# B&R Automation Studio project test
Automation Studio 4.2.5.388

## Logical view

Binary libraries used (declarations not repeated): operator, runtime, astime, AsIecCon, standard

### Global.var - Global variables
```iecst
VAR
	var2 : BOOL;
	var3 : BOOL;
	var4 : BOOL;
	var1 : BOOL;
END_VAR
```


### Program Logical/Program (IEC)

#### Cyclic.fbd - Cyclic code
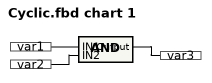
Diagram, in the editor's own instruction-list form stored in the file:
```il
PROGRAM _CYCLIC
VAR
	zz0000FCT_1_1_AND_Output : ANY;
END_VAR

{NetworkNumber := 1}
LD var1
AND var2
ST zz0000FCT_1_1_AND_Output
LD zz0000FCT_1_1_AND_Output
ST var3

END_PROGRAM
```

#### Init.fbd - Initialization code
```iecst
PROGRAM _INIT

(* TODO : Add your code here *)

END_PROGRAM
```

### dev1.txt
```
is it dev branch?
yes!
```

Listed in the project but not available here: Logical/Global.typ, Logical/Program/Exit.fbd, Logical/Program/Types.typ, Logical/Program/Variables.var
